TYPE FeederSimulation :
STRUCT
	i : INT;
END_STRUCT
END_TYPE

(* stored: Version 1.1.0.1, ProductVersion 3.1.4024.12
   DUT FeederSimulation: Id {f7e9363c-a34b-458e-aaa8-6cd49b1bd9ca} *)
